FUNCTION_BLOCK SludgeDischargeOCSLB (* CAT Function Block Type *)
  (* Standard: 61499-2 *)
  (* Version 1.2, 9/30/2026, Claude/Hidryco, Schneider Electric, Rev1.2 - Bomba disponivel = Ready OU Running; Rev1.1 - Valvula disponivel = Ready OU Aberta; Rev1 - OC6 so com nivel disponivel *)
  PACKAGE SE.Nereda;
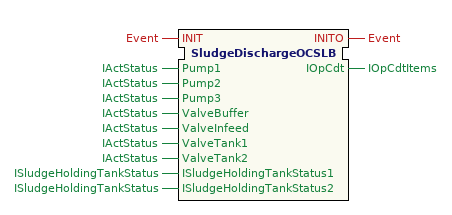
  EVENT_INPUT
    INIT;
  END_EVENT
  EVENT_OUTPUT
    INITO;
  END_EVENT
  SOCKETS
    Pump1 : IActStatus;
    Pump2 : IActStatus;
    Pump3 : IActStatus;
    ValveBuffer : IActStatus;
    ValveInfeed : IActStatus;
    ValveTank1 : IActStatus;
    ValveTank2 : IActStatus;
    ISludgeHoldingTankStatus1 : ISludgeHoldingTankStatus;
    ISludgeHoldingTankStatus2 : ISludgeHoldingTankStatus;
  END_SOCKETS
  PLUGS
    IOpCdt : IOpCdtItems;
  END_PLUGS
  (* 01 - FUNCTIONNAL INPUT INTERFACE *)
  (* 00 - INITIALIZATION *)
  (* 05 - LOGIC *)
  (* 06 - HMI INTERFACE *)
  (* 03 - FIELD INTERFACE *)
  (* 02 - FUNCTIONNAL OUTPUT INTERFACE *)
  (* Operating Condition Status *)
  (* Operating conditions : 1. Valve Tank1 OR Tank2 is available 2. Pump1 or Pump 2 or Pump 3 is available 3. Valve Buffer is closed 4. Reserved, do not use 5. Valve Infeed is closed 6. No H Level, HH at switchone Holding tank 7. Reserved 8. Both Level available *)
  FBS
    OC : encodeIOpCdt(pin_9BB2492C130556E4 := TRUE, pin_98DAA682915D8859 := TRUE, pin_6256EDBBA25FB904 := TRUE, pin_AB11CBA8876EF395 := TRUE, pin_FEDC2CE1C6BE541E := TRUE, pin_AE09A9D851459BF0 := TRUE, pin_670D03E74723DB48 := TRUE, pin_070EA4527BA3BBA8 := TRUE, pin_3B99B9D48C97D7D2 := TRUE, pin_47969CBC2D520AAD := TRUE); (* You set the operating conditions. For the inputs that are not used set a constant to TRUE. *)
    IThis : SludgeDischargeOCSLB_HMI(QI := TRUE);
    ValveTank1_OR_ValveTank2_Alvailable_1 : OR_88A3DD8EC65DD11C; {SET_ATTRIBUTE(Configuration.GenericFBType.InterfaceParams, Runtime.Standard#CNT:=2;OUT:BOOL)}
    No_Fail_No_Alarm_lt_004 : NOT_42C76073DCEB1A7A; {SET_ATTRIBUTE(Configuration.GenericFBType.InterfaceParams, Runtime.Standard#CNT:=1;OUT${CNT$}:BOOL)}
    Pum_1_2_3_Available_2 : OR_550FE6D62F509EB3; {SET_ATTRIBUTE(Configuration.GenericFBType.InterfaceParams, Runtime.Standard#CNT:=3;OUT:BOOL)}
    NoCond1 : NOT_425622A9A4AC6C60; {SET_ATTRIBUTE(Configuration.GenericFBType.InterfaceParams, Runtime.Standard#CNT:=2;OUT${CNT$}:BOOL,BOOL)}
    NoCond2 : NOT_425622A9A4AC6C60; {SET_ATTRIBUTE(Configuration.GenericFBType.InterfaceParams, Runtime.Standard#CNT:=2;OUT${CNT$}:BOOL,BOOL)}
    No_H_007 : AND_88A3DD8EC65DD11C; {SET_ATTRIBUTE(Configuration.GenericFBType.InterfaceParams, Runtime.Standard#CNT:=2;OUT:BOOL)}
    No_H_008 : AND_88A3DD8EC65DD11C; {SET_ATTRIBUTE(Configuration.GenericFBType.InterfaceParams, Runtime.Standard#CNT:=2;OUT:BOOL)}
    Both_available_008 : OR_88A3DD8EC65DD11C; {SET_ATTRIBUTE(Configuration.GenericFBType.InterfaceParams, Runtime.Standard#CNT:=2;OUT:BOOL)}
    AND1 : AND_88A3DD8EC65DD11C; {SET_ATTRIBUTE(Configuration.GenericFBType.InterfaceParams, Runtime.Standard#CNT:=2;OUT:BOOL)}
    NotAvailable : NOT_425622A9A4AC6C60; {SET_ATTRIBUTE(Configuration.GenericFBType.InterfaceParams, Runtime.Standard#CNT:=2;OUT${CNT$}:BOOL,BOOL)}
    Tank2_Ok_Or_NotAvailable : OR_88A3DD8EC65DD11C; {SET_ATTRIBUTE(Configuration.GenericFBType.InterfaceParams, Runtime.Standard#CNT:=2;OUT:BOOL)}
    Tank1_Ok_Or_NotAvailable : OR_88A3DD8EC65DD11C; {SET_ATTRIBUTE(Configuration.GenericFBType.InterfaceParams, Runtime.Standard#CNT:=2;OUT:BOOL)}
    ValveTank1_Available : OR_88A3DD8EC65DD11C; {SET_ATTRIBUTE(Configuration.GenericFBType.InterfaceParams, Runtime.Standard#CNT:=2;OUT:BOOL)}
    ValveTank2_Available : OR_88A3DD8EC65DD11C; {SET_ATTRIBUTE(Configuration.GenericFBType.InterfaceParams, Runtime.Standard#CNT:=2;OUT:BOOL)}
    Pump1_Available : OR_88A3DD8EC65DD11C; {SET_ATTRIBUTE(Configuration.GenericFBType.InterfaceParams, Runtime.Standard#CNT:=2;OUT:BOOL)}
    Pump2_Available : OR_88A3DD8EC65DD11C; {SET_ATTRIBUTE(Configuration.GenericFBType.InterfaceParams, Runtime.Standard#CNT:=2;OUT:BOOL)}
    Pump3_Available : OR_88A3DD8EC65DD11C; {SET_ATTRIBUTE(Configuration.GenericFBType.InterfaceParams, Runtime.Standard#CNT:=2;OUT:BOOL)}
  END_FBS
  EVENT_CONNECTIONS
    INIT TO IThis.26A6FDDA838D580B;
    OC.6FF8E5BE2D132B85 TO IThis.F1E666A16B4E137C;
    IThis.BC48A9191816124A TO OC.7689825C23C7E3C1;
    No_Fail_No_Alarm_lt_004.CNF TO OC.C4A26A2931936C6C;
    OC.E74FDFC5C9E17061 TO OC.C4A26A2931936C6C;
    OC.E74FDFC5C9E17061 TO INITO;
    Pump3.14377629A1F197A9 TO Pump3_Available.REQ;
    Pump2.14377629A1F197A9 TO Pump2_Available.REQ;
    Pump1.14377629A1F197A9 TO Pump1_Available.REQ;
    ValveTank1.14377629A1F197A9 TO ValveTank1_Available.REQ;
    ValveTank2.14377629A1F197A9 TO ValveTank2_Available.REQ;
    ValveInfeed.14377629A1F197A9 TO OC.C4A26A2931936C6C;
    ValveBuffer.14377629A1F197A9 TO OC.C4A26A2931936C6C;
    Pum_1_2_3_Available_2.CNF TO OC.C4A26A2931936C6C;
    ISludgeHoldingTankStatus2.903FCADE660A71D1 TO NoCond1.REQ;
    ISludgeHoldingTankStatus1.903FCADE660A71D1 TO NoCond2.REQ;
    NoCond1.CNF TO No_H_007.REQ;
    NoCond2.CNF TO No_H_008.REQ;
    ISludgeHoldingTankStatus1.903FCADE660A71D1 TO Both_available_008.REQ;
    ISludgeHoldingTankStatus2.903FCADE660A71D1 TO Both_available_008.REQ;
    Both_available_008.CNF TO OC.C4A26A2931936C6C;
    ValveTank1_OR_ValveTank2_Alvailable_1.CNF TO OC.C4A26A2931936C6C;
    AND1.CNF TO OC.C4A26A2931936C6C;
    ISludgeHoldingTankStatus1.903FCADE660A71D1 TO NotAvailable.REQ;
    ISludgeHoldingTankStatus2.903FCADE660A71D1 TO NotAvailable.REQ;
    No_H_007.CNF TO Tank2_Ok_Or_NotAvailable.REQ;
    NotAvailable.CNF TO Tank2_Ok_Or_NotAvailable.REQ;
    No_H_008.CNF TO Tank1_Ok_Or_NotAvailable.REQ;
    NotAvailable.CNF TO Tank1_Ok_Or_NotAvailable.REQ;
    Tank1_Ok_Or_NotAvailable.CNF TO AND1.REQ;
    Tank2_Ok_Or_NotAvailable.CNF TO AND1.REQ;
    ValveTank1_Available.CNF TO ValveTank1_OR_ValveTank2_Alvailable_1.REQ;
    ValveTank2_Available.CNF TO ValveTank1_OR_ValveTank2_Alvailable_1.REQ;
    Pump1_Available.CNF TO Pum_1_2_3_Available_2.REQ;
    Pump2_Available.CNF TO Pum_1_2_3_Available_2.REQ;
    Pump3_Available.CNF TO Pum_1_2_3_Available_2.REQ;
  END_CONNECTIONS
  DATA_CONNECTIONS
    OC.8E1CFBA3B24DC461 TO IThis.3DB7059599B53BF0;
    ValveTank1_OR_ValveTank2_Alvailable_1.OUT TO OC.22A84A30EE8DD605;
    ValveTank1_Available.OUT TO ValveTank1_OR_ValveTank2_Alvailable_1.IN1;
    ValveTank2_Available.OUT TO ValveTank1_OR_ValveTank2_Alvailable_1.IN2;
    Pump1_Available.OUT TO Pum_1_2_3_Available_2.IN1;
    Pump2_Available.OUT TO Pum_1_2_3_Available_2.IN2;
    Pump3_Available.OUT TO Pum_1_2_3_Available_2.IN3;
    Pum_1_2_3_Available_2.OUT TO OC.4ED40FD24D2392DA;
    ValveBuffer.3A653A8838D163CA TO OC.504E64E2CDCF5D86;
    ValveInfeed.3A653A8838D163CA TO OC.9D55FD7AD1246DA2;
    ISludgeHoldingTankStatus2.E7029D0CFFA0BD1B TO NoCond1.IN1;
    ISludgeHoldingTankStatus2.DEE031011FEE6E40 TO NoCond1.IN2;
    ISludgeHoldingTankStatus1.E7029D0CFFA0BD1B TO NoCond2.IN1;
    ISludgeHoldingTankStatus1.DEE031011FEE6E40 TO NoCond2.IN2;
    NoCond1.OUT1 TO No_H_007.IN1;
    NoCond1.OUT2 TO No_H_007.IN2;
    Tank2_Ok_Or_NotAvailable.OUT TO AND1.IN2;
    NoCond2.OUT2 TO No_H_008.IN2;
    NoCond2.OUT1 TO No_H_008.IN1;
    Tank1_Ok_Or_NotAvailable.OUT TO AND1.IN1;
    ISludgeHoldingTankStatus2.CD00A1E724699AB6 TO Both_available_008.IN1;
    ISludgeHoldingTankStatus1.CD00A1E724699AB6 TO Both_available_008.IN2;
    Both_available_008.OUT TO OC.2D24E9AB41BE5BDB;
    AND1.OUT TO OC.4E3CFAB7818DC81F;
    ISludgeHoldingTankStatus2.CD00A1E724699AB6 TO NotAvailable.IN1;
    ISludgeHoldingTankStatus1.CD00A1E724699AB6 TO NotAvailable.IN2;
    NotAvailable.OUT1 TO Tank2_Ok_Or_NotAvailable.IN1;
    No_H_007.OUT TO Tank2_Ok_Or_NotAvailable.IN2;
    NotAvailable.OUT2 TO Tank1_Ok_Or_NotAvailable.IN1;
    No_H_008.OUT TO Tank1_Ok_Or_NotAvailable.IN2;
    ValveTank1.9E0B44559326BEAF TO ValveTank1_Available.IN1;
    ValveTank1.72E790857420193D TO ValveTank1_Available.IN2;
    ValveTank2.9E0B44559326BEAF TO ValveTank2_Available.IN1;
    ValveTank2.72E790857420193D TO ValveTank2_Available.IN2;
    Pump1.9E0B44559326BEAF TO Pump1_Available.IN1;
    Pump1.D41A46B14EF7208D TO Pump1_Available.IN2;
    Pump2.9E0B44559326BEAF TO Pump2_Available.IN1;
    Pump2.D41A46B14EF7208D TO Pump2_Available.IN2;
    Pump3.9E0B44559326BEAF TO Pump3_Available.IN1;
    Pump3.D41A46B14EF7208D TO Pump3_Available.IN2;
  END_CONNECTIONS
  ADAPTER_CONNECTIONS
    OC.8E4A3B210A8341FD TO IOpCdt;
  END_CONNECTIONS
END_FUNCTION_BLOCK
